FUNCTION_BLOCK SKILL_BFB (* Basic Function Block Type *)
  (* Standard: 61499-2 *)
  (* Version 0.0, 20/04/2023, midxav, Schneider Electric, Template *)
  PACKAGE Main;
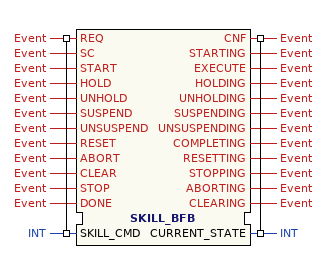
  EVENT_INPUT
    REQ WITH SKILL_CMD;
    SC;
    START;
    HOLD;
    UNHOLD;
    SUSPEND;
    UNSUSPEND;
    RESET;
    ABORT;
    CLEAR;
    STOP;
    DONE;
  END_EVENT
  EVENT_OUTPUT
    CNF WITH CURRENT_STATE;
    STARTING;
    EXECUTE;
    HOLDING;
    UNHOLDING;
    SUSPENDING;
    UNSUSPENDING;
    COMPLETING;
    RESETTING;
    STOPPING;
    ABORTING;
    CLEARING;
  END_EVENT
  VAR_INPUT
    SKILL_CMD : INT;
  END_VAR
  VAR_OUTPUT
    CURRENT_STATE : INT;
  END_VAR
  EC_STATES
    START; (* Initial State *)
    IDLE_STATE : IDLE_STATE -> CNF;
    STARTING : STARTNG -> CNF, CLEAR -> STARTING;
    EXECUTE : EXECUTE -> CNF, CLEAR -> EXECUTE;
    COMPLETING : COMPLETING -> CNF, CLEAR -> COMPLETING;
    COMPLETE : COMPLETE -> CNF;
    HOLDING : HOLDING -> CNF, CLEAR -> HOLDING;
    HELD : HELD -> CNF;
    UNHOLDING : UNHOLDING -> CNF, CLEAR -> UNHOLDING;
    SUSPENDING : SUSPENDING -> CNF, CLEAR -> SUSPENDING;
    SUSPENDED : SUSPENDED -> CNF;
    UNSUSPENDING : UNSUSPENDING -> CNF, CLEAR -> UNSUSPENDING;
    ABORTING : ABORTING -> CNF, CLEAR -> ABORTING;
    ABORTED : ABORTED -> CNF;
    CLEARING : CLEARING -> CNF, CLEAR -> CLEARING;
    STOPPING : STOPPING -> CNF, CLEAR -> STOPPING;
    STOPPED_STATE : STOPPED_STATE -> CNF;
    RESETTING : RESETTING -> CNF, CLEAR -> RESETTING;
  END_STATES
  EC_TRANSITIONS
    START TO IDLE_STATE := 1;
    IDLE_STATE TO STARTING := START OR REQ[SKILL_CMD = 1];
    STARTING TO EXECUTE := SC;
    EXECUTE TO COMPLETING := SC;
    COMPLETING TO COMPLETE := DONE;
    EXECUTE TO HOLDING := HOLD OR REQ[SKILL_CMD = 3];
    HOLDING TO HELD := SC;
    HELD TO UNHOLDING := UNHOLD OR REQ[SKILL_CMD = 4];
    UNHOLDING TO EXECUTE := SC;
    EXECUTE TO SUSPENDING := SUSPEND OR REQ[SKILL_CMD = 5];
    SUSPENDING TO SUSPENDED := SC;
    SUSPENDED TO UNSUSPENDING := UNSUSPEND OR REQ[SKILL_CMD = 6];
    UNSUSPENDING TO EXECUTE := SC;
    COMPLETE TO RESETTING := RESET OR REQ[SKILL_CMD = 2];
    ABORTING TO ABORTED := SC;
    ABORTED TO CLEARING := CLEAR OR REQ[SKILL_CMD = 7];
    CLEARING TO STOPPED_STATE := SC;
    STOPPING TO STOPPED_STATE := SC;
    STOPPED_STATE TO RESETTING := RESET OR REQ[SKILL_CMD = 2];
    RESETTING TO IDLE_STATE := SC;
    EXECUTE TO ABORTING := ABORT OR REQ[SKILL_CMD = 9];
    EXECUTE TO STOPPING := STOP OR REQ[SKILL_CMD = 8];
    STARTING TO STOPPING := REQ AND SKILL_CMD = 8;
    STOPPING TO ABORTING := ABORT OR REQ[SKILL_CMD = 9];
    CLEARING TO ABORTING := ABORT OR REQ[SKILL_CMD = 9];
  END_TRANSITIONS
  ALGORITHM IDLE_STATE IN ST:
CURRENT_STATE:= 1;
  END_ALGORITHM
  ALGORITHM STARTNG IN ST:
CURRENT_STATE:= 2;
  END_ALGORITHM
  ALGORITHM EXECUTE IN ST:
CURRENT_STATE:= 3;
  END_ALGORITHM
  ALGORITHM HOLDING IN ST:
CURRENT_STATE:=7;
  END_ALGORITHM
  ALGORITHM HELD IN ST:
CURRENT_STATE:= 8;
  END_ALGORITHM
  ALGORITHM UNHOLDING IN ST:
CURRENT_STATE:= 9;
  END_ALGORITHM
  ALGORITHM SUSPENDING IN ST:
CURRENT_STATE:= 10;
  END_ALGORITHM
  ALGORITHM SUSPENDED IN ST:
CURRENT_STATE:= 11;
  END_ALGORITHM
  ALGORITHM UNSUSPENDING IN ST:
CURRENT_STATE:= 12;
  END_ALGORITHM
  ALGORITHM COMPLETE IN ST:
CURRENT_STATE:= 5;
  END_ALGORITHM
  ALGORITHM RESETTING IN ST:
CURRENT_STATE:= 6;
  END_ALGORITHM
  ALGORITHM ABORTING IN ST:
CURRENT_STATE:= 15;
  END_ALGORITHM
  ALGORITHM ABORTED IN ST:
CURRENT_STATE:= 16;
  END_ALGORITHM
  ALGORITHM CLEARING IN ST:
CURRENT_STATE:= 17;
  END_ALGORITHM
  ALGORITHM STOPPING IN ST:
CURRENT_STATE:= 13;
  END_ALGORITHM
  ALGORITHM STOPPED_STATE IN ST:
CURRENT_STATE:= 14;
  END_ALGORITHM
  ALGORITHM COMPLETING IN ST:
CURRENT_STATE:= 4;
  END_ALGORITHM
  ALGORITHM CLEAR IN ST:
SC := FALSE;
  END_ALGORITHM
END_FUNCTION_BLOCK
